PROGRAM MAIN
VAR

END_VAR


GantryRobotMotion();
PLC_PRG();

END_PROGRAM

(* stored: Version 1.1.0.1, ProductVersion 3.1.4022.12
   POU MAIN: Id {104ec441-47eb-4139-a2a2-70833eb8a567}, SpecialFunc None *)
